PROGRAM FocusControl
VAR_INPUT
	// enable the axis
	enable: BOOL;
	// Move M2 closer to M1
	inward: 	BOOL;
	// Move M2 away from M1
	outward: 	BOOL;	
	// reset the axis(-error)
	reset: 		BOOL;
	// move the axis to new position
	MoveAxis:	BOOL;
	// calibrate the focus axis
	HomeAxis:	BOOL;
	// focus position in millimeters
	position: 		LREAL;
END_VAR

VAR_OUTPUT
	// true if absolute calibration
	Calibrated:	BOOL;
	// true if error
	Error: 		BOOL;
	// ID of NC axis error
	ErrorID:	UDINT;
	// ready signal = drive ready + standstill
	Ready:	BOOL;
END_VAR

VAR
	FocusDelay:			TON;
	FocusAxis:			FB_Axis2;
	actual_position:	LREAL;
	Focus_max:			LREAL;
	FocusUnlock:		BOOL;
	FocusUnlocked:		BOOL;
	FocusCalibration:	MC_SetPosition;
	MQTTTimer : 		TON := (PT:=T#5S);
	getlastposition:	BOOL := TRUE;
	FocusAxisEvent:		FB_EventLog;
	CalibrationEvent:	FB_EventLog;
END_VAR

VAR CONSTANT
	// reference position for homing
	homing_position:		LREAL := 97.96; // 107,50 - 9,54
	calibration_position:	LREAL := 0.0;
	tolerance:				LREAL := 0.001;
END_VAR
VAR PERSISTENT
	last_position:	LREAL := -1.0;
END_VAR

(*
Focus Control Unit
spindle gear: 5mm
brake: 86 61103H00 Var. 0005 Index C; 24VDC geglattet 0,25 A P1672/R7
motor: Faulhaber ; Schönaich ; 3557K024CR; 454  431 ; Made in germany ==> 5300 rpm
gear: Faulhaber ; MINIMOTOR SA ; swiss made ; 38/1S  43:1 ; 033896  503
Focus is locked by default
*)

GVL_Telescope.focus_unlock := enable AND NOT FocusAxis.StandStill;

// wait until the focus is unlocked for n milliseconds
FocusDelay(IN := GVL_Telescope.focus_unlock, PT := T#500MS, Q => FocusUnlocked);

IF HomeAxis THEN
	position := homing_position;
END_IF

// deactivate limit switches on homing
MC_SetAcceptBlockedDriveSignal(
	Axis := GVL_Telescope.FocusAxisRef, 
	Enable := HomeAxis);

//GVL_Telescope.focus_lock := FocusUnlocked;
FocusAxis(	
	Enable := 			enable,
	Reset := 			reset,
	MoveAxis := 		MoveAxis,
	HomeAxis :=			HomeAxis,
	Position := 		position,
	Velocity :=			1.0,
	Enable_Positive := 	NOT GVL_Telescope.focus_limit_far OR HomeAxis,
	Enable_Negative := 	NOT GVL_Telescope.focus_limit_near,
	Jog_Forward :=		outward,
	Jog_Backwards := 	inward,
	bCalibrationCam :=  GVL_Telescope.focus_limit_far,
	ActualPosition => 	actual_position,
	Error =>			error,
	ErrorID =>			ErrorID,
	AxisRef :=			GVL_Telescope.FocusAxisRef);	

IF FocusAxis.MoveDone THEN
	MoveAxis := FALSE;
END_IF

IF FocusAxis.HomeDone THEN
	HomeAxis := FALSE;
END_IF
	
IF FocusAxis.ResetDone THEN
	reset := FALSE;
END_IF

IF FocusAxis.Calibrated OR Error THEN
	HomeAxis := FALSE;
END_IF

Calibrated := FocusAxis.Calibrated;

IF getlastposition AND last_position>=0.0 AND NOT Calibrated THEN
	// calibrate on stored position
	FocusCalibration.Execute := getlastposition AND FocusAxis.Ready;
	FocusCalibration.Position := last_position;
ELSE
	// Calibrate on near end
	FocusCalibration.Execute := GVL_Telescope.focus_limit_near;
	FocusCalibration.Position := calibration_position;
END_IF
	

FocusCalibration(Axis := GVL_Telescope.FocusAxisRef);

IF FocusCalibration.Done OR Calibrated THEN
	last_position := actual_position;
	getlastposition := FALSE;
END_IF

	
IF GVL_Telescope.focus_limit_far THEN
	Focus_max := actual_position;
END_IF

IF Calibrated AND ABS(actual_position - position) > tolerance THEN
	MoveAxis := TRUE;
ELSE
	MoveAxis := FALSE;
END_IF

Ready := FocusAxis.Ready AND FocusAxis.StandStill;

MQTTTimer(IN:=Enable);
IF MQTTTimer.Q THEN // publish new payload every second
	MQTTTimer(IN:=FALSE);
	MAIN.MQTTClient.Publish('telescope', 'dome', 'FocusPosition', LREAL_TO_FMTSTR(actual_position, 5, TRUE));
	MAIN.MQTTClient.Publish('telescope', 'dome', 'FocusCalibrated', BOOL_TO_STRING(Calibrated));	
	MAIN.MQTTClient.Publish('telescope', 'dome', 'FocusReady', BOOL_TO_STRING(Ready));	
	
END_IF

FocusAxisEvent(	
	Trigger := 		FocusAxis.Error, 
	Level := 		ADSLOG_MSGTYPE_ERROR,
	FormatString :=	'Focus Axis Error: %s',
	OnMessage := 	NCError_TO_STRING(ErrorID),
	OffMEssage := 	'OK',
	OffLevel := 	ADSLOG_MSGTYPE_HINT);

CalibrationEvent(
	Trigger :=	Calibrated,
	Level :=	ADSLOG_MSGTYPE_HINT,
	OnMessage := 'Focus is calibrated.'
	);

END_PROGRAM

(* stored: Version 1.1.0.1, ProductVersion 3.1.4024.9
   POU FocusControl: Id {d08d0458-4211-4cc5-9e25-2b5c152fb2d4}, SpecialFunc None *)
